TYPE ST_UserManagment :
STRUCT
	userID 				:	INT;			//numer porządkowy użytkownika
//	domain				:	STRING(80);
	enabled				:	BOOL;
	userLogin			:	STRING(80);		//login do zalogowania
	userNameSurname 	:	WSTRING(255);	//imię i nazwisko
	userNameSurnameNumber	:UINT;
	password			:	STRING(255);	//hasło kalwiaturowe
	passwordRFID		:	STRING(255);	//hasło rfid
	passwordQR			:	STRING(255);	//hasło qr
	userGroup			:	STRING(80);		//grupa użytkowników
	userGropuNumber		:	UINT;			//numer grupy
//	autoLogOff			:	STRING(80);		//czas do wylogowania
//	locale				:	STRING(80);		//gdzie zapisujemy
//	timeFormatlocale	:	STRING(80);		//format godziny
//	timeZone			:	STRING(80);		//strefa czasowa
	signedPassword		:	STRING(80);		//hasło przekazywane do HMI
END_STRUCT
END_TYPE

(* stored: Version 1.1.0.1, ProductVersion 3.1.4026.13, FileIdentifier 8f1e5ecd5750c44fb0f848e7133696eb425cbe04, FileSignature 65cbc5ecc99194211a8bbee7c2089ac63c828b81fc040a8ad0f59ea2af9aaae30c7e101723a60f59626e2fb9523d2bc7d19f3e45871461ba1fd83e75a962e35482e4435e4f8e305d5306efb5efaa0ddf78e76bd6d858c0cb8dbf9d80d820aed6af415709edb216a64859378cc22623548e792545eca26fa084c37ae912e13f2556cbd6c747ba30c9bfd50f8c7cf051a506ca29440133550dd0bf6ded4dad14fc2e64e26bb575f582a5003c56c06cc0d9b0cadd1a16ce57b8c97aba03842b2363e4869dceaafd7245f72762049f67560c14035f2b9844b3c44c482c29859f54e7d87bc36e714c9ee08849ff3c5395328168a3a0523a4ddb76690d67e24c11216c
   DUT ST_UserManagment: Id {cd6a86f3-3b0d-4eb8-9588-d25443aab3ee} *)
